FUNCTION_BLOCK FB_Loader
VAR_INPUT
	EN : BOOL;
	Level_Prox : BOOL; // Loader Proximity Switch
	Flap_Reed : BOOL; // Loader Flap Reed Switch
	Switch : BOOL; // Loader switch
	PushButton : BOOL; // Loader Push Button
	Vac_Grant : BOOL; // Vacuum Grant to the Loader
	Switch_Bit : BOOL; // Loader internal Switch Bit - Push Button or Switch
END_VAR
VAR_OUTPUT
	ENO : BOOL;
	Valve : BOOL; // Loader Vacuum Valve
	Lamp : BOOL; // Loader status lamp
	Comp_Status : WORD; // Loader status word for Sysmetric Vision
	HMI_Status : WORD; // Loader status word for HMI
	Vac_Request : BOOL; // Vacuum Request from the loader
END_VAR
VAR
	tempTimer1 : TON;
	tempTimer2 : TON;
	Timer0_5_s : TON;
	MATfallTIME : CTU;
	Flap_Open_time : CTU;
	CONValarm : CTU;
	One_Time : BOOL;
	Switch_Keep : SR;
END_VAR
VAR // added by the converter: edge detectors and wires of the graphical bodies
    _rt1, _rt2 : R_TRIG;
    _ft1 : F_TRIG;
    _w1, _w2, _w3 : BOOL;
END_VAR

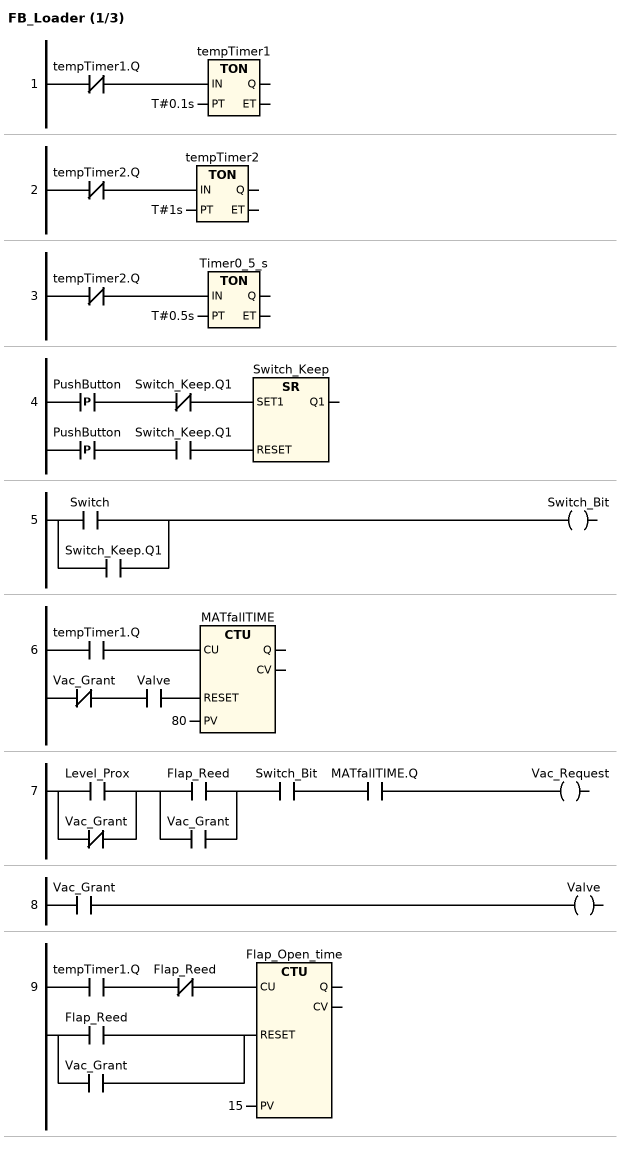
// NETWORK 1
tempTimer1(IN := NOT tempTimer1.Q, PT := T#0.1s); // TON

// NETWORK 2
tempTimer2(IN := NOT tempTimer2.Q, PT := T#1s); // TON

// NETWORK 3
Timer0_5_s(IN := NOT tempTimer2.Q, PT := T#0.5s); // TON

// NETWORK 4
_rt1(CLK := PushButton);
_rt2(CLK := PushButton);
Switch_Keep(SET1 := _rt1.Q AND NOT Switch_Keep.Q1, RESET := _rt2.Q AND Switch_Keep.Q1); // SR

// NETWORK 5
Switch_Bit := Switch OR Switch_Keep.Q1;

// NETWORK 6
MATfallTIME(CU := tempTimer1.Q, RESET := NOT Vac_Grant AND Valve, PV := 80); // CTU

// NETWORK 7
Vac_Request := (Level_Prox OR NOT Vac_Grant) AND (Flap_Reed OR Vac_Grant) AND Switch_Bit AND MATfallTIME.Q;

// NETWORK 8
Valve := Vac_Grant;

// NETWORK 9
Flap_Open_time(CU := tempTimer1.Q AND NOT Flap_Reed, RESET := Flap_Reed OR Vac_Grant, PV := 15); // CTU

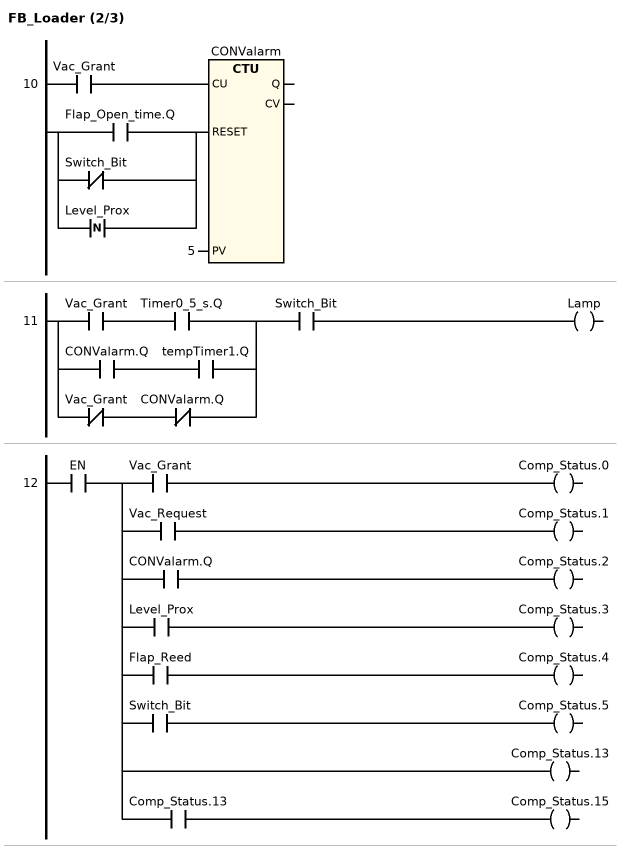
// NETWORK 10
_ft1(CLK := Level_Prox);
CONValarm(CU := Vac_Grant, RESET := Flap_Open_time.Q OR NOT Switch_Bit OR _ft1.Q, PV := 5); // CTU

// NETWORK 11
Lamp := (Vac_Grant AND Timer0_5_s.Q OR CONValarm.Q AND tempTimer1.Q OR NOT Vac_Grant AND NOT CONValarm.Q) AND Switch_Bit;

// NETWORK 12
Comp_Status.0 := EN AND Vac_Grant;
Comp_Status.1 := EN AND Vac_Request;
Comp_Status.2 := EN AND CONValarm.Q;
Comp_Status.3 := EN AND Level_Prox;
Comp_Status.4 := EN AND Flap_Reed;
Comp_Status.5 := EN AND Switch_Bit;
Comp_Status.13 := EN;
Comp_Status.15 := EN AND Comp_Status.13;

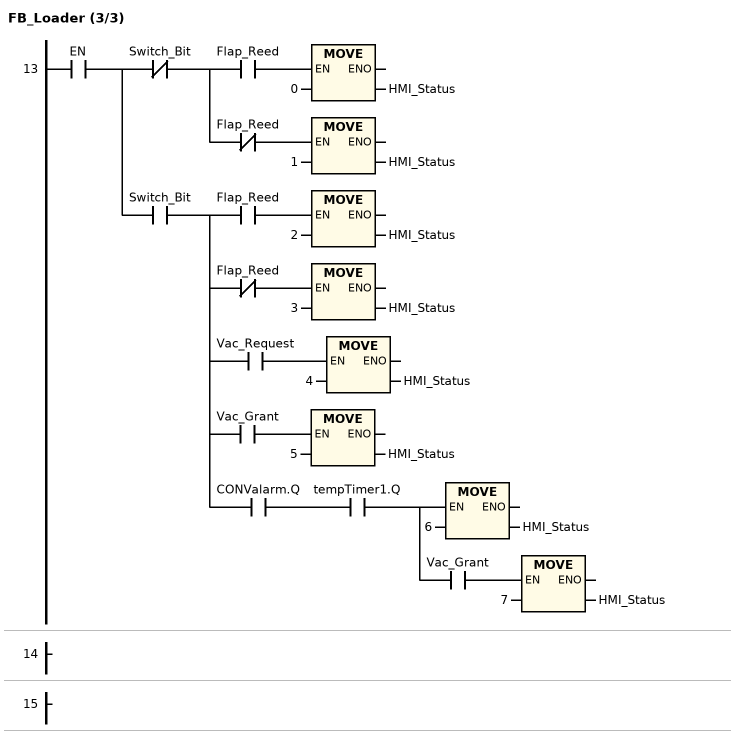
// NETWORK 13
_w1 := EN AND NOT Switch_Bit;
IF _w1 AND Flap_Reed THEN HMI_Status := 0; END_IF
IF _w1 AND NOT Flap_Reed THEN HMI_Status := 1; END_IF
_w2 := EN AND Switch_Bit;
IF _w2 AND Flap_Reed THEN HMI_Status := 2; END_IF
IF _w2 AND NOT Flap_Reed THEN HMI_Status := 3; END_IF
IF _w2 AND Vac_Request THEN HMI_Status := 4; END_IF
IF _w2 AND Vac_Grant THEN HMI_Status := 5; END_IF
_w3 := _w2 AND CONValarm.Q AND tempTimer1.Q;
IF _w3 THEN HMI_Status := 6; END_IF
IF _w3 AND Vac_Grant THEN HMI_Status := 7; END_IF

// NETWORK 14

// NETWORK 15

END_FUNCTION_BLOCK

(* stored: Version 1.1.0.1, ProductVersion 3.1.4024.13
   POU FB_Loader: Id {81e6a8e4-985e-48e1-92ce-6cdaa989c6d8}, SpecialFunc None *)
